FUNCTION TFFuoriIngombroVerticaleOK : BOOL
VAR_INPUT
	QuotaAsseZ : LREAL;
	Mission : POINTER TO TFMachinePalletizer_Mission;
END_VAR
VAR
END_VAR

(* Controllo Asse Z Fuori Ingombro *)
CASE Mission^.TPick OF
	TPICK_LAYER:
					IF QuotaAsseZ >= QuotaFuoriIngombro_Z_AVUOTO OR 
					QuotaAsseZ >= QuotaFuoriIngombro_Z_ConFALDA THEN
						TFFuoriIngombroVerticaleOK := TRUE;
					ELSE
						TFFuoriIngombroVerticaleOK := FALSE;
					END_IF
	TPICK_PACK :
					IF QuotaAsseZ >= QuotaFuoriIngombro_Z_AVUOTO OR 
					QuotaAsseZ >= QuotaFuoriIngombro_Z_ConPEZZO THEN
						TFFuoriIngombroVerticaleOK := TRUE;
					ELSE
						TFFuoriIngombroVerticaleOK := FALSE;
					END_IF
	TPICK_PALLET:
					IF QuotaAsseZ >= QuotaFuoriIngombro_Z_AVUOTO OR 
					QuotaAsseZ >= QuotaFuoriIngombro_Z_ConPALLET THEN
						TFFuoriIngombroVerticaleOK := TRUE;
					ELSE
						TFFuoriIngombroVerticaleOK := FALSE;
					END_IF
					
	TPICK_NOT_DEFINED:
					IF QuotaAsseZ >= QuotaFuoriIngombro_Z_AVUOTO OR 
					QuotaAsseZ >= QuotaFuoriIngombro_Z_ConPEZZO OR 
					QuotaAsseZ >= QuotaFuoriIngombro_Z_ConPALLET OR
					QuotaAsseZ >= QuotaFuoriIngombro_Z_ConFALDA THEN
						TFFuoriIngombroVerticaleOK := TRUE;
					ELSE
						TFFuoriIngombroVerticaleOK := FALSE;
					END_IF
					
	TPICK_LASTRA:
					IF QuotaAsseZ >= QuotaFuoriIngombro_Z_AVUOTO OR 
					QuotaAsseZ >= QuotaFuoriIngombro_Z_ConPEZZO THEN
						TFFuoriIngombroVerticaleOK := TRUE;
					ELSE
						TFFuoriIngombroVerticaleOK := FALSE;
					END_IF
					
	TPICK_QUADROTTA:
					IF QuotaAsseZ >= QuotaFuoriIngombro_Z_AVUOTO OR 
					QuotaAsseZ >= QuotaFuoriIngombro_Z_ConPEZZO THEN
						TFFuoriIngombroVerticaleOK := TRUE;
					ELSE
						TFFuoriIngombroVerticaleOK := FALSE;
					END_IF
					
					
					
					
					
END_CASE

END_FUNCTION

(* stored: Version 1.1.0.1, ProductVersion 3.1.4024.11
   POU TFFuoriIngombroVerticaleOK: Id {04056c1e-a816-4242-a546-74a651eaf43a}, SpecialFunc None *)
